# EPICS autosave request: iocBoot/iocxxx/scan1Menu.req
file configMenu.req P=$(P),CONFIG=$(CONFIG)
file scan_settings.req P=$(P),S=scan2
file scan_settings.req P=$(P),S=scan1
file scan_settings.req P=$(P),S=scanH
